// TIA Portal V20 export
// export: Created 2026-07-12T13:33:04.873902Z, ExportSetting WithDefaults, DisplayName Totally Integrated Automation Portal, DisplayVersion V20 Update 4, DisplayName TIA Portal Openness, DisplayVersion V20 Update 4, DisplayName TIA Portal Version Control Interface, DisplayVersion V20 Update 4, DisplayName STEP 7 Professional, DisplayVersion V20 Update 4, DisplayName STEP 7 Safety, DisplayVersion V20 Update 2, DisplayName WinCC Basic/Comfort/Advanced, DisplayVersion V20 Update 4, DisplayName WinCC Unified, DisplayVersion V20 Update 4
DATA_BLOCK "DB_Test"   // DB7
{ S7_Optimized_Access := 'FALSE' }
VERSION : 0.1
// stored: AutoNumber true, IsOnlyStoredInLoadMemory false, IsWriteProtectedInAS false
   VAR RETAIN
      Saw1 : Bool;
      Saw2 : Bool;
      Saw3 : Bool;
      Saw4 : Bool;
      Saw5 : Bool;
      Saw6 : Bool;
      Saw7 : Bool;
      Saw8 : Bool;
      Saw9 : Bool;
      Saw10 : Bool;
      SawDown : Bool;
      ProflefromSelection : Word;
      OrginSimulation : Bool;
      ThicknessSimulation : Real;
      ProxySim : Bool;
      StartMachineSimulation : Bool;
      ProxyCountSimulation : DInt;
      L_CutlineSensorSim : Array[1..15] of Bool;
      B_ManipButtonsSim : Array[1..15] of Bool;
      Reset_ExceptionSim : Bool;
      Reset_Buffer : Bool;
   END_VAR
BEGIN
END_DATA_BLOCK
